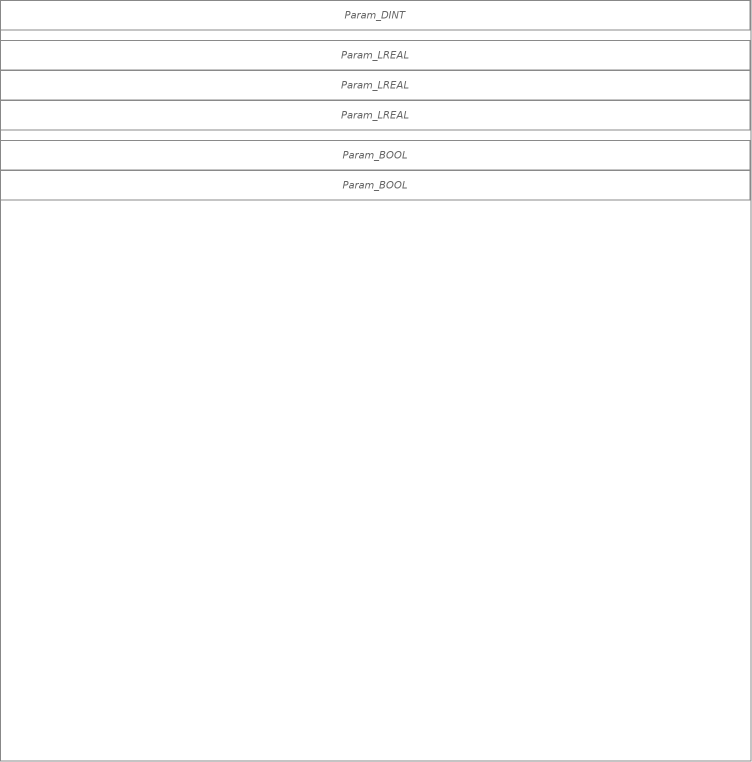
VISUALIZATION Visu_Mparam_Supply  // 752x762
    Frame (0,40 750x30)
        shows Param_LREAL(nIdx := 21)
    Frame (0,70 750x30)
        shows Param_LREAL(nIdx := 22)
    Frame (0,100 750x30)
        shows Param_LREAL(nIdx := 23)
    Frame (0,0 750x30)
        shows Param_DINT(nIdx := 6)
    Frame (0,140 750x30)
        shows Param_BOOL(nIdx := 11)
    Frame (0,170 750x30)
        shows Param_BOOL(nIdx := 15)
    Rectangle (0,730 750x30)
END_VISUALIZATION

(* stored: Version 1.1.0.1, ProductVersion 3.1.4024.12
   Visu Visu_Mparam_Supply: Id {2a3c611d-f10a-4d00-96f6-7ea3aa3831ff} *)
